KUKA KRL data list: sbt_comm003.dat

&ACCESS RVEO
defdat sbt_comm003 public
;***********************************************************
;
; file Name: sbt_comm003
;
; Description:
;   Language             ==   KRL for KUKA ROBOT
;   Date                 ==   2024 - 06 - 03
;   Modification Data    ==   2022 - 06 - 03
;
; Author: speedbot
;
; Version: 1.0
;***********************************************************


decl cmd_typ01_t CmdType01
decl cmd_typ03_t CmdType03
decl int Status                        = 0
decl pos CurPos                                                                           ; 存储当前直角坐标坐标



enddat
